VAR_GLOBAL
	Digital_Output AT %Q* : ARRAY [1..10] OF BOOL;
END_VAR

(* stored: Version 1.1.0.1, ProductVersion 3.1.0.36
   GVL IO_DigiOut_GVL: Id {de4775a9-03ff-4acb-85b8-047d20026ef0} *)
